(*
Description: 
Interface that every function block that wants to be a subscriber, needs to implement.
*)
INTERFACE I_SubCallback

(*
Description: 
the callback that will be invoked when there is a publish for what the subscriber was subscribed to.
*)
METHOD Callback
VAR_INPUT
	data : PubSubData;
END_VAR
END_METHOD

END_INTERFACE

(* stored: Version 1.1.0.1, ProductVersion 3.1.4024.12
   Itf I_SubCallback: Id {02583392-d99a-4331-aea4-211798062edf}
   Method Callback: Id {51ae99f5-b00c-4730-906a-01e66248c5b3} *)
